ABB RAPID module: Module1.mod

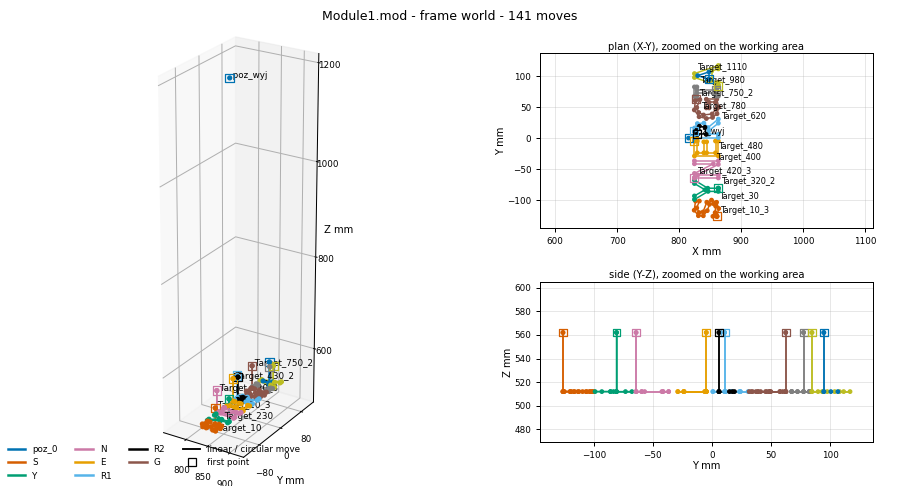
[picture p0: tool path of Module1.mod in frame world, 141 of 141 moves have a stored position in this frame; points joined in program order, loops and branches not executed]
MODULE Module1
    CONST robtarget poz_wyj:=[[815,0,1186.5],[0,0,1,0],[0,0,0,0],[9E9,9E9,9E9,9E9,9E9,9E9]];
    CONST robtarget Target_10:=[[1060.644210049,-141.073722293,462.000385148],[0.000000116,0.222660799,0.974895978,0.000000322],[-1,0,-1,1],[9E9,9E9,9E9,9E9,9E9,9E9]];
    CONST robtarget Target_20:=[[1063.63892504,-128.437479389,461.999793984],[-0.000000098,0.22266118,0.974895891,-0.000000116],[-1,0,-1,1],[9E9,9E9,9E9,9E9,9E9,9E9]];
    CONST robtarget Target_30:=[[1060.144970722,-118.391852583,461.999735622],[-0.000000316,0.22266118,0.974895891,0.000000052],[-1,0,-1,1],[9E9,9E9,9E9,9E9,9E9,9E9]];
    CONST robtarget Target_40:=[[1051.970864374,-114.8973241,461.999954041],[-0.000000233,0.22266118,0.974895891,-0.000000011],[-1,0,-1,1],[9E9,9E9,9E9,9E9,9E9,9E9]];
    CONST robtarget Target_50:=[[1044.365911594,-118.291619091,461.999686424],[-0.000000235,0.22266118,0.974895891,-0.000000133],[-1,0,-1,1],[9E9,9E9,9E9,9E9,9E9,9E9]];
    CONST robtarget Target_60:=[[1038.32204036,-133.987056543,461.999993919],[0.000000099,0.22266118,0.974895891,-0.000000015],[-1,0,-1,1],[9E9,9E9,9E9,9E9,9E9,9E9]];
    CONST robtarget Target_70:=[[1032.042989466,-135.023435002,462.000508776],[0.000000268,0.22266118,0.974895891,0.000000277],[-1,0,-1,1],[9E9,9E9,9E9,9E9,9E9,9E9]];
    CONST robtarget Target_80:=[[1028.196976193,-127.501358358,461.99958652],[-0.000000347,0.22266118,0.974895891,-0.000000313],[-1,0,-1,1],[9E9,9E9,9E9,9E9,9E9,9E9]];
    CONST robtarget Target_90:=[[1032.377938839,-116.394513212,462.000172264],[0.000000035,0.22266118,0.974895891,0.000000235],[-1,0,-1,1],[9E9,9E9,9E9,9E9,9E9,9E9]];
    CONST robtarget Target_100:=[[1026.262857713,-116.394957654,462.000007987],[-0.00000004,0.22266118,0.974895891,0.000000063],[-1,0,-1,1],[9E9,9E9,9E9,9E9,9E9,9E9]];
    CONST robtarget Target_110:=[[1032.377938839,-116.394513212,462.000172264],[0.000000035,0.22266059,0.974896026,0.000000235],[-1,0,-1,1],[9E9,9E9,9E9,9E9,9E9,9E9]];
    CONST robtarget Target_120:=[[1026.262857713,-116.394957654,462.000007987],[-0.00000004,0.222660726,0.974895995,0.000000063],[-1,0,-1,1],[9E9,9E9,9E9,9E9,9E9,9E9]];
    CONST robtarget Target_130:=[[1024.079108629,-131.19555289,461.999801728],[0.000000003,0.22266118,0.974895891,-0.000000047],[-1,0,-1,1],[9E9,9E9,9E9,9E9,9E9,9E9]];
    CONST robtarget Target_140:=[[1030.836019059,-140.037978755,462.000063071],[-0.000000118,0.22266118,0.974895891,0.000000173],[-1,0,-1,1],[9E9,9E9,9E9,9E9,9E9,9E9]];
    CONST robtarget Target_150:=[[1038.775878877,-140.124225855,461.999694483],[-0.00000041,0.222660658,0.97489601,0.000000172],[-1,0,-1,1],[9E9,9E9,9E9,9E9,9E9,9E9]];
    CONST robtarget Target_160:=[[1045.137948073,-131.932343429,462.000377039],[0.000000218,0.222660786,0.974895981,0.000000033],[-1,0,-1,1],[9E9,9E9,9E9,9E9,9E9,9E9]];
    CONST robtarget Target_170:=[[1048.676727604,-121.689567913,462.000176875],[0.000000014,0.222660561,0.974896033,-0.000000117],[-1,0,-1,1],[9E9,9E9,9E9,9E9,9E9,9E9]];
    CONST robtarget Target_180:=[[1055.443307497,-120.79553311,462.000382561],[0.000000304,0.222660904,0.974895954,0.000000194],[-1,0,-1,1],[9E9,9E9,9E9,9E9,9E9,9E9]];
    CONST robtarget Target_190:=[[1058.58378636,-124.494250783,461.999632746],[-0.000000198,0.22266085,0.974895967,-0.000000234],[-1,0,-1,1],[9E9,9E9,9E9,9E9,9E9,9E9]];
    CONST robtarget Target_200:=[[1057.899095188,-134.974131209,462.000232536],[0.000000209,0.222660682,0.974896005,-0.000000189],[-1,0,-1,1],[9E9,9E9,9E9,9E9,9E9,9E9]];
    CONST robtarget Target_210:=[[1054.216635753,-141.073965467,461.999499526],[-0.000000397,0.22266118,0.974895891,0.000000297],[-1,0,-1,1],[9E9,9E9,9E9,9E9,9E9,9E9]];
    CONST robtarget Target_10_2:=[[1060.644210049,-141.073722293,462.000385148],[0.000000116,0.22266118,0.974895891,0.000000322],[-1,0,-1,1],[9E9,9E9,9E9,9E9,9E9,9E9]];
    CONST robtarget Target_220:=[[1062.952976122,-95.740877551,462.000031118],[-0.000000014,0.222661188,0.97489589,-0.000000017],[0,0,-1,1],[9E9,9E9,9E9,9E9,9E9,9E9]];
    CONST robtarget Target_230:=[[1045.917873668,-95.741393135,462.000189003],[0.000000162,0.22266157,0.974895802,0.000000128],[0,0,-1,1],[9E9,9E9,9E9,9E9,9E9,9E9]];
    CONST robtarget Target_240:=[[1024.452841566,-82.731235578,462.00012578],[-0.000000027,0.222661506,0.974895817,-0.000000207],[0,0,-1,1],[9E9,9E9,9E9,9E9,9E9,9E9]];
    CONST robtarget Target_250:=[[1024.452815737,-88.159602261,461.999721931],[-0.00000034,0.222661323,0.974895859,-0.000000198],[0,0,-1,1],[9E9,9E9,9E9,9E9,9E9,9E9]];
    CONST robtarget Target_260:=[[1041.393949358,-98.267508726,461.999600438],[-0.000000333,0.222660771,0.974895985,-0.000000042],[0,0,-1,1],[9E9,9E9,9E9,9E9,9E9,9E9]];
    CONST robtarget Target_270:=[[1024.453259029,-108.188997559,462.000666672],[0.000000466,0.222660945,0.974895945,0.000000158],[-1,0,-1,1],[9E9,9E9,9E9,9E9,9E9,9E9]];
    CONST robtarget Target_290:=[[1024.453264391,-113.867272151,462.000343494],[0.000000039,0.222660854,0.974895966,0.000000118],[-1,0,-1,1],[9E9,9E9,9E9,9E9,9E9,9E9]];
    CONST robtarget Target_300:=[[1046.447998744,-100.857062099,461.999708121],[-0.000000201,0.222660755,0.974895988,-0.000000095],[0,0,-1,1],[9E9,9E9,9E9,9E9,9E9,9E9]];
    CONST robtarget Target_310:=[[1062.952852921,-100.857822025,461.99982389],[-0.000000052,0.222661369,0.974895848,-0.000000342],[0,0,-1,1],[9E9,9E9,9E9,9E9,9E9,9E9]];
    CONST robtarget Target_320:=[[1062.952910873,-95.741201482,461.999821712],[-0.00000025,0.222661408,0.974895839,-0.000000071],[0,0,-1,1],[9E9,9E9,9E9,9E9,9E9,9E9]];
    CONST robtarget Target_420:=[[1024.452922061,-79.174027693,462],[0,0.222660835,0.97489597,0],[0,0,-1,1],[9E9,9E9,9E9,9E9,9E9,9E9]];
    CONST robtarget Target_410:=[[1024.452922061,-71.904578926,462],[0,0.222660835,0.97489597,0],[0,0,-1,1],[9E9,9E9,9E9,9E9,9E9,9E9]];
    CONST robtarget Target_400:=[[1054.934687919,-56.398501514,462],[0,0.222660835,0.97489597,0],[0,0,-1,1],[9E9,9E9,9E9,9E9,9E9,9E9]];
    CONST robtarget Target_390:=[[1024.452922061,-56.398501514,462],[0,0.222660835,0.97489597,0],[0,0,-1,1],[9E9,9E9,9E9,9E9,9E9,9E9]];
    CONST robtarget Target_380:=[[1024.452922061,-51.625000822,462],[0,0.222660835,0.97489597,0],[0,0,-1,1],[9E9,9E9,9E9,9E9,9E9,9E9]];
    CONST robtarget Target_370:=[[1062.952921108,-51.625000822,462],[0,0.222660835,0.97489597,0],[0,0,-1,1],[9E9,9E9,9E9,9E9,9E9,9E9]];
    CONST robtarget Target_360:=[[1062.952921108,-57.365681393,462],[0,0.222660835,0.97489597,0],[0,0,-1,1],[9E9,9E9,9E9,9E9,9E9,9E9]];
    CONST robtarget Target_350:=[[1029.756811719,-74.400527,462],[0,0.222660835,0.97489597,0],[0,0,-1,1],[9E9,9E9,9E9,9E9,9E9,9E9]];
    CONST robtarget Target_340:=[[1062.952921108,-74.400527,462],[0,0.222660835,0.97489597,0],[0,0,-1,1],[9E9,9E9,9E9,9E9,9E9,9E9]];
    CONST robtarget Target_330:=[[1062.952921108,-79.174027693,462],[0,0.222660835,0.97489597,0],[0,0,-1,1],[9E9,9E9,9E9,9E9,9E9,9E9]];
    CONST robtarget Target_420_2:=[[1024.452922061,-79.174027693,462],[0,0.222660835,0.97489597,0],[0,0,-1,1],[9E9,9E9,9E9,9E9,9E9,9E9]];
    CONST robtarget Target_430:=[[1024.452922061,-19.739264173,462],[0,0.222660835,0.97489597,0],[0,0,-1,1],[9E9,9E9,9E9,9E9,9E9,9E9]];
    CONST robtarget Target_440:=[[1024.452922061,-43.82516309,462],[0,0.222660835,0.97489597,0],[0,0,-1,1],[9E9,9E9,9E9,9E9,9E9,9E9]];
    CONST robtarget Target_450:=[[1062.952921108,-43.82516309,462],[0,0.222660835,0.97489597,0],[0,0,-1,1],[9E9,9E9,9E9,9E9,9E9,9E9]];
    CONST robtarget Target_460:=[[1062.952921108,-19.739264173,462],[0,0.222660835,0.97489597,0],[0,0,-1,1],[9E9,9E9,9E9,9E9,9E9,9E9]];
    CONST robtarget Target_470:=[[1058.397815872,-19.739264173,462],[0,0.222660835,0.97489597,0],[0,0,-1,1],[9E9,9E9,9E9,9E9,9E9,9E9]];
    CONST robtarget Target_480:=[[1058.397815872,-38.708469538,462],[0,0.222660835,0.97489597,0],[0,0,-1,1],[9E9,9E9,9E9,9E9,9E9,9E9]];
    CONST robtarget Target_490:=[[1044.108513146,-38.708469538,462],[0,0.222660835,0.97489597,0],[0,0,-1,1],[9E9,9E9,9E9,9E9,9E9,9E9]];
    CONST robtarget Target_500:=[[1044.108513146,-21.018437561,462],[0,0.222660835,0.97489597,0],[0,0,-1,1],[9E9,9E9,9E9,9E9,9E9,9E9]];
    CONST robtarget Target_510:=[[1039.553407911,-21.018437561,462],[0,0.222660835,0.97489597,0],[0,0,-1,1],[9E9,9E9,9E9,9E9,9E9,9E9]];
    CONST robtarget Target_520:=[[1039.553407911,-38.708469538,462],[0,0.222660835,0.97489597,0],[0,0,-1,1],[9E9,9E9,9E9,9E9,9E9,9E9]];
    CONST robtarget Target_530:=[[1029.008027297,-38.708469538,462],[0,0.222660835,0.97489597,0],[0,0,-1,1],[9E9,9E9,9E9,9E9,9E9,9E9]];
    CONST robtarget Target_540:=[[1029.008027297,-19.739264173,462],[0,0.222660835,0.97489597,0],[0,0,-1,1],[9E9,9E9,9E9,9E9,9E9,9E9]];
    CONST robtarget Target_550:=[[1024.452922061,-19.739264173,462],[0,0.222660835,0.97489597,0],[0,0,-1,1],[9E9,9E9,9E9,9E9,9E9,9E9]];
    CONST robtarget Target_560:=[[1024.452922061,-4.20198741,462],[0,0.222660835,0.97489597,0],[0,0,-1,1],[9E9,9E9,9E9,9E9,9E9,9E9]];
    CONST robtarget Target_570:=[[1024.452922061,-14.123381006,462],[0,0.222660835,0.97489597,0],[0,0,-1,1],[9E9,9E9,9E9,9E9,9E9,9E9]];
    CONST robtarget Target_580:=[[1062.952921108,-14.123381006,462],[0,0.222660835,0.97489597,0],[0,0,-1,1],[9E9,9E9,9E9,9E9,9E9,9E9]];
    CONST robtarget Target_590:=[[1062.952921108,-9.006687453,462],[0,0.222660835,0.97489597,0],[0,0,-1,1],[9E9,9E9,9E9,9E9,9E9,9E9]];
    CONST robtarget Target_600:=[[1047.634039801,-9.006687453,462],[0,0.222660835,0.97489597,0],[0,0,-1,1],[9E9,9E9,9E9,9E9,9E9,9E9]];
    CONST robtarget Target_610:=[[1047.634039801,-3.141209479,462],[0,0.222660835,0.97489597,0],[0,0,-1,1],[9E9,9E9,9E9,9E9,9E9,9E9]];
    CONST robtarget Target_620:=[[1062.952921108,9.026537384,462],[0,0.222660835,0.97489597,0],[0,0,-1,1],[9E9,9E9,9E9,9E9,9E9,9E9]];
    CONST robtarget Target_630:=[[1062.952921108,15.671999131,462],[0,0.222660835,0.97489597,0],[0,0,-1,1],[9E9,9E9,9E9,9E9,9E9,9E9]];
    CONST robtarget Target_640:=[[1046.198869659,1.975484074,462],[0,0.222660835,0.97489597,0],[0,0,-1,1],[9E9,9E9,9E9,9E9,9E9,9E9]];
    CONST robtarget Target_650:=[[1039.694735167,9.099301132,462],[0,0.222660835,0.97489597,0],[0,0,-1,1],[9E9,9E9,9E9,9E9,9E9,9E9]];
    CONST robtarget Target_660:=[[1029.15950648,8.368800445,462],[0,0.222660835,0.97489597,0],[0,0,-1,1],[9E9,9E9,9E9,9E9,9E9,9E9]];
    CONST robtarget Target_670:=[[1024.811714597,1.33589738,462],[0,0.222660835,0.97489597,0],[0,0,-1,1],[9E9,9E9,9E9,9E9,9E9,9E9]];
    CONST robtarget Target_680:=[[1024.452922061,-4.20198741,462],[0,0.222660835,0.97489597,0],[0,0,-1,1],[9E9,9E9,9E9,9E9,9E9,9E9]];
    CONST robtarget Target_690:=[[1028.883229893,-9.006687453,462],[0,0.222661369,0.974895848,0],[0,0,-1,1],[9E9,9E9,9E9,9E9,9E9,9E9]];
    CONST robtarget Target_700:=[[1043.359728724,-9.006687453,462],[0,0.222661369,0.974895848,0],[0,0,-1,1],[9E9,9E9,9E9,9E9,9E9,9E9]];
    CONST robtarget Target_710:=[[1041.362970265,2.443474338,462],[0,0.222661369,0.974895848,0],[0,0,-1,1],[9E9,9E9,9E9,9E9,9E9,9E9]];
    CONST robtarget Target_720:=[[1032.534240483,4.123148634,462],[0,0.222661369,0.974895848,0],[0,0,-1,1],[9E9,9E9,9E9,9E9,9E9,9E9]];
    CONST robtarget Target_730:=[[1029.225283131,-0.138351644,462],[0,0.222661369,0.974895848,0],[0,0,-1,1],[9E9,9E9,9E9,9E9,9E9,9E9]];
    CONST robtarget Target_740:=[[1028.883229893,-9.006687453,462],[0,0.222661369,0.974895848,0],[0,0,-1,1],[9E9,9E9,9E9,9E9,9E9,9E9]];
    CONST robtarget Target_750:=[[1027.073667539,47.495337079,462],[0,0.222661369,0.974895848,0],[0,0,-1,1],[9E9,9E9,9E9,9E9,9E9,9E9]];
    CONST robtarget Target_760:=[[1033.251139023,47.058546166,462],[0,0.222661369,0.974895848,0],[0,0,-1,1],[9E9,9E9,9E9,9E9,9E9,9E9]];
    CONST robtarget Target_770:=[[1028.196844173,34.298011636,462],[0,0.222661369,0.974895848,0],[0,0,-1,1],[9E9,9E9,9E9,9E9,9E9,9E9]];
    CONST robtarget Target_780:=[[1031.341145776,26.261272447,462],[0,0.222661369,0.974895848,0],[0,0,-1,1],[9E9,9E9,9E9,9E9,9E9,9E9]];
    CONST robtarget Target_790:=[[1039.099789798,22.278538468,462],[0,0.222661369,0.974895848,0],[0,0,-1,1],[9E9,9E9,9E9,9E9,9E9,9E9]];
    CONST robtarget Target_800:=[[1052.961328973,23.893028101,462],[0,0.222661369,0.974895848,0],[0,0,-1,1],[9E9,9E9,9E9,9E9,9E9,9E9]];
    CONST robtarget Target_810:=[[1058.932478457,31.524550784,462],[0,0.222661369,0.974895848,0],[0,0,-1,1],[9E9,9E9,9E9,9E9,9E9,9E9]];
    CONST robtarget Target_820:=[[1058.023423661,42.597038983,462],[0,0.222661369,0.974895848,0],[0,0,-1,1],[9E9,9E9,9E9,9E9,9E9,9E9]];
    CONST robtarget Target_830:=[[1048.070830714,42.597038983,462],[0,0.222661369,0.974895848,0],[0,0,-1,1],[9E9,9E9,9E9,9E9,9E9,9E9]];
    CONST robtarget Target_840:=[[1048.070830714,33.674024617,462],[0,0.222661369,0.974895848,0],[0,0,-1,1],[9E9,9E9,9E9,9E9,9E9,9E9]];
    CONST robtarget Target_850:=[[1043.578124181,33.674024617,462],[0,0.222661369,0.974895848,0],[0,0,-1,1],[9E9,9E9,9E9,9E9,9E9,9E9]];
    CONST robtarget Target_860:=[[1043.578124181,47.651333834,462],[0,0.222661369,0.974895848,0],[0,0,-1,1],[9E9,9E9,9E9,9E9,9E9,9E9]];
    CONST robtarget Target_870:=[[1060.394574331,47.651333834,462],[0,0.222661369,0.974895848,0],[0,0,-1,1],[9E9,9E9,9E9,9E9,9E9,9E9]];
    CONST robtarget Target_880:=[[1063.70170553,34.859599953,462],[0,0.222661369,0.974895848,0],[0,0,-1,1],[9E9,9E9,9E9,9E9,9E9,9E9]];
    CONST robtarget Target_890:=[[1060.885964108,24.24012088,462],[0,0.222661369,0.974895848,0],[0,0,-1,1],[9E9,9E9,9E9,9E9,9E9,9E9]];
    CONST robtarget Target_900:=[[1053.618785266,18.324047292,462],[0,0.222661369,0.974895848,0],[0,0,-1,1],[9E9,9E9,9E9,9E9,9E9,9E9]];
    CONST robtarget Target_910:=[[1043.671722233,16.545580957,462],[0,0.222661369,0.974895848,0],[0,0,-1,1],[9E9,9E9,9E9,9E9,9E9,9E9]];
    CONST robtarget Target_920:=[[1031.925166609,19.447120594,462],[0,0.222661369,0.974895848,0],[0,0,-1,1],[9E9,9E9,9E9,9E9,9E9,9E9]];
    CONST robtarget Target_930:=[[1024.223657624,30.391997136,462],[0,0.222661369,0.974895848,0],[0,0,-1,1],[9E9,9E9,9E9,9E9,9E9,9E9]];
    CONST robtarget Target_940:=[[1025.888092204,44.936990303,462],[0,0.222661369,0.974895848,0],[0,0,-1,1],[9E9,9E9,9E9,9E9,9E9,9E9]];
    CONST robtarget Target_950:=[[1027.073667539,47.495337079,462],[0,0.222661369,0.974895848,0],[0,0,-1,1],[9E9,9E9,9E9,9E9,9E9,9E9]];
    CONST robtarget Target_960:=[[1059.02180289,62.595822929,462],[0,0.222661369,0.974895848,0],[0,0,-1,1],[9E9,9E9,9E9,9E9,9E9,9E9]];
    CONST robtarget Target_970:=[[1028.384040278,62.595822929,462],[0,0.222661369,0.974895848,0],[0,0,-1,1],[9E9,9E9,9E9,9E9,9E9,9E9]];
    CONST robtarget Target_980:=[[1028.384040278,67.494121024,462],[0,0.222661369,0.974895848,0],[0,0,-1,1],[9E9,9E9,9E9,9E9,9E9,9E9]];
    CONST robtarget Target_990:=[[1024.452922061,67.494121024,462],[0,0.222661369,0.974895848,0],[0,0,-1,1],[9E9,9E9,9E9,9E9,9E9,9E9]];
    CONST robtarget Target_1000:=[[1024.452922061,52.58083128,462],[0,0.222661369,0.974895848,0],[0,0,-1,1],[9E9,9E9,9E9,9E9,9E9,9E9]];
    CONST robtarget Target_1010:=[[1028.384040278,52.58083128,462],[0,0.222661369,0.974895848,0],[0,0,-1,1],[9E9,9E9,9E9,9E9,9E9,9E9]];
    CONST robtarget Target_1020:=[[1028.384040278,57.479129376,462],[0,0.222661369,0.974895848,0],[0,0,-1,1],[9E9,9E9,9E9,9E9,9E9,9E9]];
    CONST robtarget Target_1030:=[[1059.02180289,57.479129376,462],[0,0.222661369,0.974895848,0],[0,0,-1,1],[9E9,9E9,9E9,9E9,9E9,9E9]];
    CONST robtarget Target_1040:=[[1059.02180289,52.58083128,462],[0,0.222661369,0.974895848,0],[0,0,-1,1],[9E9,9E9,9E9,9E9,9E9,9E9]];
    CONST robtarget Target_1050:=[[1062.952921108,52.58083128,462],[0,0.222661369,0.974895848,0],[0,0,-1,1],[9E9,9E9,9E9,9E9,9E9,9E9]];
    CONST robtarget Target_1060:=[[1062.952921108,67.494121024,462],[0,0.222661369,0.974895848,0],[0,0,-1,1],[9E9,9E9,9E9,9E9,9E9,9E9]];
    CONST robtarget Target_1070:=[[1059.02180289,67.494121024,462],[0,0.222661369,0.974895848,0],[0,0,-1,1],[9E9,9E9,9E9,9E9,9E9,9E9]];
    CONST robtarget Target_1080:=[[1059.02180289,62.595822929,462],[0,0.222661369,0.974895848,0],[0,0,-1,1],[9E9,9E9,9E9,9E9,9E9,9E9]];
    CONST robtarget Target_1090:=[[1062.952921108,69.678075589,462],[0,0.222661369,0.974895848,0],[0,0,-1,1],[9E9,9E9,9E9,9E9,9E9,9E9]];
    CONST robtarget Target_1100:=[[1024.452922061,82.657005576,462],[0,0.222661369,0.974895848,0],[0,0,-1,1],[9E9,9E9,9E9,9E9,9E9,9E9]];
    CONST robtarget Target_1110:=[[1024.452922061,88.959274464,462],[0,0.222661369,0.974895848,0],[0,0,-1,1],[9E9,9E9,9E9,9E9,9E9,9E9]];
    CONST robtarget Target_1120:=[[1062.952921108,101.93820445,462],[0,0.222661369,0.974895848,0],[0,0,-1,1],[9E9,9E9,9E9,9E9,9E9,9E9]];
    CONST robtarget Target_1130:=[[1062.952921108,96.540716739,462],[0,0.222661369,0.974895848,0],[0,0,-1,1],[9E9,9E9,9E9,9E9,9E9,9E9]];
    CONST robtarget Target_1140:=[[1052.189145037,93.046389435,462],[0,0.222661369,0.974895848,0],[0,0,-1,1],[9E9,9E9,9E9,9E9,9E9,9E9]];
    CONST robtarget Target_1150:=[[1052.189145037,78.351495148,462],[0,0.222661369,0.974895848,0],[0,0,-1,1],[9E9,9E9,9E9,9E9,9E9,9E9]];
    CONST robtarget Target_1160:=[[1062.952921108,74.857167844,462],[0,0.222661369,0.974895848,0],[0,0,-1,1],[9E9,9E9,9E9,9E9,9E9,9E9]];
    CONST robtarget Target_1170:=[[1047.821235907,79.75546594,462],[0,0.222661369,0.974895848,0],[0,0,-1,1],[9E9,9E9,9E9,9E9,9E9,9E9]];
    CONST robtarget Target_1180:=[[1029.694413017,85.683342616,462],[0,0.222661369,0.974895848,0],[0,0,-1,1],[9E9,9E9,9E9,9E9,9E9,9E9]];
    CONST robtarget Target_1190:=[[1047.821235907,91.642418643,462],[0,0.222661369,0.974895848,0],[0,0,-1,1],[9E9,9E9,9E9,9E9,9E9,9E9]];
    CONST robtarget Target_1200:=[[1047.821235907,79.75546594,462],[0,0.222661369,0.974895848,0],[0,0,-1,1],[9E9,9E9,9E9,9E9,9E9,9E9]];
    CONST robtarget Target_10_3:=[[1060.644191571,-141.073751102,512.000385148],[0.000000116,0.22266118,0.974895891,0.000000322],[-1,0,-1,1],[9E9,9E9,9E9,9E9,9E9,9E9]];
    CONST robtarget Target_320_2:=[[1062.952936826,-95.741200127,511.999821712],[-0.00000025,0.222661408,0.974895839,-0.000000071],[0,0,-1,1],[9E9,9E9,9E9,9E9,9E9,9E9]];
    CONST robtarget Target_420_3:=[[1024.452922061,-79.174027693,512],[0,0.222660835,0.97489597,0],[0,0,-1,1],[9E9,9E9,9E9,9E9,9E9,9E9]];
    CONST robtarget Target_430_2:=[[1024.452922061,-19.739264173,512],[0,0.222660835,0.97489597,0],[0,0,-1,1],[9E9,9E9,9E9,9E9,9E9,9E9]];
    CONST robtarget Target_560_2:=[[1024.452922061,-4.20198741,512],[0,0.222660835,0.97489597,0],[0,0,-1,1],[9E9,9E9,9E9,9E9,9E9,9E9]];
    CONST robtarget Target_690_2:=[[1028.883229893,-9.006687453,512],[0,0.222661369,0.974895848,0],[0,0,-1,1],[9E9,9E9,9E9,9E9,9E9,9E9]];
    CONST robtarget Target_750_2:=[[1027.073667539,47.495337079,512],[0,0.222661369,0.974895848,0],[0,0,-1,1],[9E9,9E9,9E9,9E9,9E9,9E9]];
    CONST robtarget Target_960_2:=[[1059.02180289,62.595822929,512],[0,0.222661369,0.974895848,0],[0,0,-1,1],[9E9,9E9,9E9,9E9,9E9,9E9]];
    CONST robtarget Target_1090_2:=[[1062.952921108,69.678075589,512],[0,0.222661369,0.974895848,0],[0,0,-1,1],[9E9,9E9,9E9,9E9,9E9,9E9]];
    CONST robtarget Target_1170_2:=[[1047.821235907,79.75546594,512],[0,0.222661369,0.974895848,0],[0,0,-1,1],[9E9,9E9,9E9,9E9,9E9,9E9]];

    PROC poz_0()
        MoveJ poz_wyj,v400,fine,Pen_TCP\WObj:=wobj0;
	ENDPROC
    PROC S()
        SingArea\Wrist;
        ConfL\Off;
        MoveJ Target_10_3,v400,z1,Pen_TCP\WObj:=Sheet;
        MoveL Target_10,v300,fine,Pen_TCP\WObj:=Sheet;
        MoveL Target_20,v100,z1,Pen_TCP\WObj:=Sheet;
        MoveL Target_30,v100,z1,Pen_TCP\WObj:=Sheet;
        MoveL Target_40,v100,z1,Pen_TCP\WObj:=Sheet;
        MoveL Target_50,v100,z1,Pen_TCP\WObj:=Sheet;
        MoveL Target_60,v100,z1,Pen_TCP\WObj:=Sheet;
        MoveL Target_70,v100,z1,Pen_TCP\WObj:=Sheet;
        MoveL Target_80,v100,z1,Pen_TCP\WObj:=Sheet;
        MoveL Target_90,v100,z1,Pen_TCP\WObj:=Sheet;
        MoveL Target_100,v100,z1,Pen_TCP\WObj:=Sheet;
        MoveL Target_130,v100,z1,Pen_TCP\WObj:=Sheet;
        MoveL Target_140,v100,z1,Pen_TCP\WObj:=Sheet;
        MoveL Target_150,v100,z1,Pen_TCP\WObj:=Sheet;
        MoveL Target_160,v100,fine,Pen_TCP\WObj:=Sheet;
        MoveL Target_170,v100,z1,Pen_TCP\WObj:=Sheet;
        MoveL Target_180,v100,z1,Pen_TCP\WObj:=Sheet;
        MoveL Target_190,v100,z1,Pen_TCP\WObj:=Sheet;
        MoveL Target_200,v100,z1,Pen_TCP\WObj:=Sheet;
        MoveL Target_210,v100,z1,Pen_TCP\WObj:=Sheet;
        MoveL Target_10_2,v100,z1,Pen_TCP\WObj:=Sheet;
        MoveL Target_10_3,v300,z1,Pen_TCP\WObj:=Sheet;
    ENDPROC
    PROC Y()
        MoveL Target_320_2,v400,z1,Pen_TCP\WObj:=Sheet;
        MoveL Target_220,v300,fine,Pen_TCP\WObj:=Sheet;
        MoveL Target_230,v100,z1,Pen_TCP\WObj:=Sheet;
        MoveL Target_240,v100,z1,Pen_TCP\WObj:=Sheet;
        MoveL Target_250,v100,z1,Pen_TCP\WObj:=Sheet;
        MoveL Target_260,v100,z1,Pen_TCP\WObj:=Sheet;
        MoveL Target_270,v100,z1,Pen_TCP\WObj:=Sheet;
        MoveL Target_290,v100,z1,Pen_TCP\WObj:=Sheet;
        MoveL Target_300,v100,z1,Pen_TCP\WObj:=Sheet;
        MoveL Target_310,v100,z1,Pen_TCP\WObj:=Sheet;
        MoveL Target_320,v100,fine,Pen_TCP\WObj:=Sheet;
        MoveL Target_320_2,v300,z1,Pen_TCP\WObj:=Sheet;
    ENDPROC
    PROC N()
        MoveL Target_420_3,v400,z1,Pen_TCP\WObj:=Sheet;
        MoveL Target_420,v300,fine,Pen_TCP\WObj:=Sheet;
        MoveL Target_410,v100,z1,Pen_TCP\WObj:=Sheet;
        MoveL Target_400,v100,z1,Pen_TCP\WObj:=Sheet;
        MoveL Target_390,v100,z1,Pen_TCP\WObj:=Sheet;
        MoveL Target_380,v100,z1,Pen_TCP\WObj:=Sheet;
        MoveL Target_370,v100,z1,Pen_TCP\WObj:=Sheet;
        MoveL Target_360,v100,z1,Pen_TCP\WObj:=Sheet;
        MoveL Target_350,v100,z1,Pen_TCP\WObj:=Sheet;
        MoveL Target_340,v100,z1,Pen_TCP\WObj:=Sheet;
        MoveL Target_330,v100,z1,Pen_TCP\WObj:=Sheet;
        MoveL Target_420_2,v100,fine,Pen_TCP\WObj:=Sheet;
        MoveL Target_420_3,v300,z1,Pen_TCP\WObj:=Sheet;
    ENDPROC
    PROC E()
        MoveL Target_430_2,v400,z1,Pen_TCP\WObj:=Sheet;
        MoveL Target_430,v300,fine,Pen_TCP\WObj:=Sheet;
        MoveL Target_440,v100,z1,Pen_TCP\WObj:=Sheet;
        MoveL Target_450,v100,z1,Pen_TCP\WObj:=Sheet;
        MoveL Target_460,v100,z1,Pen_TCP\WObj:=Sheet;
        MoveL Target_470,v100,z1,Pen_TCP\WObj:=Sheet;
        MoveL Target_480,v100,z1,Pen_TCP\WObj:=Sheet;
        MoveL Target_490,v100,z1,Pen_TCP\WObj:=Sheet;
        MoveL Target_500,v100,z1,Pen_TCP\WObj:=Sheet;
        MoveL Target_510,v100,z1,Pen_TCP\WObj:=Sheet;
        MoveL Target_520,v100,z1,Pen_TCP\WObj:=Sheet;
        MoveL Target_530,v100,z1,Pen_TCP\WObj:=Sheet;
        MoveL Target_540,v100,fine,Pen_TCP\WObj:=Sheet;
        MoveL Target_550,v100,z1,Pen_TCP\WObj:=Sheet;
        MoveL Target_430_2,v300,z1,Pen_TCP\WObj:=Sheet;
    ENDPROC
    PROC R1()
        SingArea\Wrist;
        ConfL\Off;
        MoveL Target_560_2,v400,z1,Pen_TCP\WObj:=Sheet;
        MoveL Target_560,v300,fine,Pen_TCP\WObj:=Sheet;
        MoveL Target_570,v100,z1,Pen_TCP\WObj:=Sheet;
        MoveL Target_580,v100,z1,Pen_TCP\WObj:=Sheet;
        MoveL Target_590,v100,z1,Pen_TCP\WObj:=Sheet;
        MoveL Target_600,v100,z1,Pen_TCP\WObj:=Sheet;
        MoveL Target_610,v100,z1,Pen_TCP\WObj:=Sheet;
        MoveL Target_620,v100,z1,Pen_TCP\WObj:=Sheet;
        MoveL Target_630,v100,z1,Pen_TCP\WObj:=Sheet;
        MoveL Target_640,v100,z1,Pen_TCP\WObj:=Sheet;
        MoveL Target_650,v100,z1,Pen_TCP\WObj:=Sheet;
        MoveL Target_660,v100,z1,Pen_TCP\WObj:=Sheet;
        MoveL Target_670,v100,z1,Pen_TCP\WObj:=Sheet;
        MoveL Target_680,v100,fine,Pen_TCP\WObj:=Sheet;
        MoveL Target_560_2,v300,z1,Pen_TCP\WObj:=Sheet;
    ENDPROC
    PROC R2()
        SingArea\Wrist;
        ConfL\Off;
        MoveL Target_690_2,v400,z1,Pen_TCP\WObj:=Sheet;
        MoveL Target_690,v300,fine,Pen_TCP\WObj:=Sheet;
        MoveL Target_700,v100,z1,Pen_TCP\WObj:=Sheet;
        MoveL Target_710,v100,z1,Pen_TCP\WObj:=Sheet;
        MoveL Target_720,v100,z1,Pen_TCP\WObj:=Sheet;
        MoveL Target_730,v100,z1,Pen_TCP\WObj:=Sheet;
        MoveL Target_740,v100,fine,Pen_TCP\WObj:=Sheet;
        MoveL Target_690_2,v300,z1,Pen_TCP\WObj:=Sheet;
    ENDPROC
    PROC G()
        SingArea\Wrist;
        ConfL\Off;
        MoveL Target_750_2,v400,z1,Pen_TCP\WObj:=Sheet;
        MoveL Target_750,v300,fine,Pen_TCP\WObj:=Sheet;
        MoveL Target_760,v100,z1,Pen_TCP\WObj:=Sheet;
        MoveL Target_770,v100,z1,Pen_TCP\WObj:=Sheet;
        MoveL Target_780,v100,z1,Pen_TCP\WObj:=Sheet;
        MoveL Target_790,v100,z1,Pen_TCP\WObj:=Sheet;
        MoveL Target_800,v100,z1,Pen_TCP\WObj:=Sheet;
        MoveL Target_810,v100,z1,Pen_TCP\WObj:=Sheet;
        MoveL Target_820,v100,z1,Pen_TCP\WObj:=Sheet;
        MoveL Target_830,v100,z1,Pen_TCP\WObj:=Sheet;
        MoveL Target_840,v100,z1,Pen_TCP\WObj:=Sheet;
        MoveL Target_850,v100,z1,Pen_TCP\WObj:=Sheet;
        MoveL Target_860,v100,z1,Pen_TCP\WObj:=Sheet;
        MoveL Target_870,v100,z1,Pen_TCP\WObj:=Sheet;
        MoveL Target_880,v100,z1,Pen_TCP\WObj:=Sheet;
        MoveL Target_890,v100,z1,Pen_TCP\WObj:=Sheet;
        MoveL Target_900,v100,z1,Pen_TCP\WObj:=Sheet;
        MoveL Target_910,v100,z1,Pen_TCP\WObj:=Sheet;
        MoveL Target_920,v100,z1,Pen_TCP\WObj:=Sheet;
        MoveL Target_930,v100,z1,Pen_TCP\WObj:=Sheet;
        MoveL Target_940,v100,z1,Pen_TCP\WObj:=Sheet;
        MoveL Target_950,v100,fine,Pen_TCP\WObj:=Sheet;
        MoveL Target_750_2,v300,z1,Pen_TCP\WObj:=Sheet;
    ENDPROC
    PROC I()
        MoveL Target_960_2,v400,z1,Pen_TCP\WObj:=Sheet;
        MoveL Target_960,v300,fine,Pen_TCP\WObj:=Sheet;
        MoveL Target_970,v100,z1,Pen_TCP\WObj:=Sheet;
        MoveL Target_980,v100,z1,Pen_TCP\WObj:=Sheet;
        MoveL Target_990,v100,z1,Pen_TCP\WObj:=Sheet;
        MoveL Target_1000,v100,z1,Pen_TCP\WObj:=Sheet;
        MoveL Target_1010,v100,z1,Pen_TCP\WObj:=Sheet;
        MoveL Target_1020,v100,z1,Pen_TCP\WObj:=Sheet;
        MoveL Target_1030,v100,z1,Pen_TCP\WObj:=Sheet;
        MoveL Target_1040,v100,z1,Pen_TCP\WObj:=Sheet;
        MoveL Target_1050,v100,z1,Pen_TCP\WObj:=Sheet;
        MoveL Target_1060,v100,z1,Pen_TCP\WObj:=Sheet;
        MoveL Target_1070,v100,z1,Pen_TCP\WObj:=Sheet;
        MoveL Target_1080,v100,fine,Pen_TCP\WObj:=Sheet;
        MoveL Target_960_2,v300,z1,Pen_TCP\WObj:=Sheet;
    ENDPROC
    PROC A1()
        MoveL Target_1090_2,v400,z1,Pen_TCP\WObj:=Sheet;
        MoveL Target_1090,v300,fine,Pen_TCP\WObj:=Sheet;
        MoveL Target_1100,v100,z1,Pen_TCP\WObj:=Sheet;
        MoveL Target_1110,v100,z1,Pen_TCP\WObj:=Sheet;
        MoveL Target_1120,v100,z1,Pen_TCP\WObj:=Sheet;
        MoveL Target_1130,v100,z1,Pen_TCP\WObj:=Sheet;
        MoveL Target_1140,v100,z1,Pen_TCP\WObj:=Sheet;
        MoveL Target_1150,v100,z1,Pen_TCP\WObj:=Sheet;
        MoveL Target_1160,v100,z1,Pen_TCP\WObj:=Sheet;
        MoveL Target_1090,v100,fine,Pen_TCP\WObj:=Sheet;
        MoveL Target_1090_2,v300,z1,Pen_TCP\WObj:=Sheet;
    ENDPROC
    PROC A2()
        MoveL Target_1170_2,v400,z1,Pen_TCP\WObj:=Sheet;
        MoveL Target_1170,v300,fine,Pen_TCP\WObj:=Sheet;
        MoveL Target_1180,v100,z1,Pen_TCP\WObj:=Sheet;
        MoveL Target_1190,v100,z1,Pen_TCP\WObj:=Sheet;
        MoveL Target_1200,v100,fine,Pen_TCP\WObj:=Sheet;
        MoveL Target_1170_2,v300,z1,Pen_TCP\WObj:=Sheet;
    ENDPROC
    PROC rDoExit()
        STOP;
    ENDPROC

ENDMODULE
